PROGRAM MAIN
VAR
	p1, p2 : Piston;

END_VAR

p1(delay := T#2S, timeout := T#4S, pistonName := 'linear1');
p2(delay := T#2S, timeout := T#4S, pistonName := 'drawer2');

END_PROGRAM

(* stored: Version 1.1.0.1, ProductVersion 3.1.4022.18
   POU MAIN: Id {d7a22d48-d601-42e4-8b6f-48cd53a4aca2}, SpecialFunc None *)
